(* IEC 61131-3 sources: eCockpitGit/test_project/src/%F%00 Library/%F%Common Functions/%F%Networking/%POU%FB_TCPMultiPlexer/%PRO%messageHandler, 2 files *)

(* ---- %GETSET%Get.st ---- *)
VAR
END_VAR

(*%!%__DELIMITER__%!%*)
messageHandler			:=		S_messageEvent;

(* ---- %GETSET%Set.st ---- *)
VAR
	i		:WORD;
END_VAR

(*%!%__DELIMITER__%!%*)
S_messageEvent							:=		messageHandler;
IF S_controllersSize > 0 THEN
	FOR i := 0 TO S_controllersSize - 1 DO
		S_controllers^[i].S_message		:=		S_messageEvent;
	END_FOR
END_IF
